{attribute 'qualified_only'}
{attribute 'strict'}
TYPE E_OperationMode : // Operation modes defined
(
	Initialization :=1,
	Service :=2,
	Manual :=3,
	Simulation :=4,
	Automatic :=5
);
END_TYPE

(* stored: Version 1.1.0.1, ProductVersion 3.1.4024.6
   EnumerationTextList E_OperationMode: Id {cc27e6c4-e77d-4b70-b735-d13484b5d06e} *)
